Fanuc KAREL source: kt00055.KL

-- PROVISIONAL review KL for V1013-1; original PC SHA256 ad74d51e9acb3f68a52d8e10f9792b62b8b62fa204777d703c016385a30bac19
-- Incomplete behavior may be omitted. Consult companion uncertainty JSON. Do not deploy.
PROGRAM KT00055
%NOLOCKGROUP
VAR
  OUT : INTEGER
-- UNRESOLVED_DECL Y1 type=002018
-- UNRESOLVED_DECL H2 type=002017
BEGIN
  -- UNRESOLVED_PC offsets 5-19; opcodes 2E,22,9D,33,B2
  -- UNRESOLVED_PC offsets 24-38; opcodes 2E,22,9D,33,B4
  -- UNRESOLVED_PC offsets 43-68; opcodes 22,9D,33,B1,22,9D,33,B3,53,23
  -- UNRESOLVED_PC offsets 73-77; opcodes 7F
END KT00055
